// TIA Portal V16 export
// export: Created 2021-05-26T11:33:08.319044Z, ExportSetting WithDefaults, DisplayName Totally Integrated Automation Portal, DisplayVersion V16 Update 4, DisplayName TIA Portal Version Control Interface, DisplayVersion V16 Update 2, DisplayName TIA Portal Openness, DisplayVersion V16 Update 4, DisplayName STEP 7 Professional, DisplayVersion V16 Update 4, DisplayName STEP 7 Safety, DisplayVersion V16, DisplayName WinCC Advanced, DisplayVersion V16 Update 4
ORGANIZATION_BLOCK "Check_EthernetCommun"   // OB31, STL, CyclicInterrupt
{ S7_Optimized_Access := 'TRUE' }
VERSION : 0.1
// Project:   CRE-331M  SSA PLC control system
// Copyright: 2020 Cryoelectra GmbH
// Purpose:Control UDP communication between Mikrocontrollers and PLC
// Versions:  
// 0.0  18-Feb-2020  fam  initial version                                  00
// 0.1   23-Jun-2020  fam  added fan controllers                   01
// 0.2   24-Jul-2020   bam  added warnings handling          02
// stored: AutoNumber true
   VAR_INPUT
      Initial_Call : Bool;   // Initial call of this OB
      Event_Count : Int;   // Events discarded
   END_VAR
BEGIN

NETWORK
TITLE = 01
//      CALL  "FC_COMM_ModCon10"   //debug

      CALL  "FC_checkCommUDP";

      CALL  "FC_checkCommFanCons";

      CALL  "FC_WarningsHandling";  //02


END_ORGANIZATION_BLOCK
